(* Logix 5000 project; controller cal1632 1756-L62 rev 16.20; software revision 16.05; part 4 of 57 *)
(* tags used below, declared in another part *)
   FAULT : BOOL;
   HMI : BOOL;
   p01_ai_prs : REAL;
   p01_ai_tc : REAL;
   p01_di_edge_ctrl_estop_active : BOOL;
   p01_di_estop_1_tripped : BOOL;
   p01_di_estop_2_tripped : BOOL;
   p01_di_estop_reset : BOOL;
   p01_di_impreg_estop_active : BOOL;
   p01_di_letoff_estop_active : BOOL;
   p01_di_lof_acc_estop_active : BOOL;
   p01_di_main_hmi_estop : BOOL;
   p01_di_rope_sw_1_active : BOOL;
   p01_di_rope_sw_2_active : BOOL;
   p01_di_rope_sw_3_active : BOOL;
   p01_di_rope_sw_4_active : BOOL;
   p01_di_rope_sw_5_active : BOOL;
   p01_di_rope_sw_6_active : BOOL;
   p01_di_rope_sw_7_active : BOOL;
   p01_di_rope_sw_8_active : BOOL;
   p01_di_splice_estop_active : BOOL;
   p01_di_ts2_estop_active : BOOL;
   p01_di_winder_estop_active : BOOL;
   p01_dint_to_hmi : DINT[16];
   p01_int_from_oxidizer : INT[10];
   p01_param_master_jog_speed : REAL;
   p01_real_to_hmi : REAL[112];
   p01r02 : routine;
   p01r02_all_fans_stopped : BOOL;
   p01r02_batch_run_time_hrs : DINT;
   p01r02_do_horn : BOOL;
   p01r02_horn : BOOL;
   p01r02_timer_half_second_on : TIMER;
   p01r02_timer_second : TIMER[2];
   p01r03 : routine;
   p01r03_oxidizer_prs : SYS_SCP;
   p01r03_prs_input_max : REAL;
   p01r03_prs_input_min : REAL;
   p01r03_prs_output_max : REAL;
   p01r03_prs_output_min : REAL;
   p01r03_timer_fault : TIMER[4];
   p01r03_timer_warning : TIMER[4];
   p01r04 : routine;
   p01r04_LFL_warning : BOOL;
   p01r04_Temp_deviation_warning : BOOL;
   p01r04_timer_fault : TIMER[4];
   p01r04_timer_warning : TIMER[4];
   p01r05 : routine;
   p01r05_enc : SYS_ENC;
   p01r05_timer_fault : TIMER[4];
   p01r05_timer_warning : TIMER[4];
   p01r06 : routine;
   p01r06_timer_fault : TIMER[4];
   p01r06_timer_warning : TIMER[4];
   p01r07 : routine;
   p01r07_timer_fault : TIMER[4];
   p01r07_timer_warning : TIMER[4];
   p01r09 : routine;
   p01r09_mode_jog : BOOL;
   p01r09_mode_run : BOOL;
   p01r09_mode_thread : BOOL;
   p01r09_open_oven : BOOL;
   p01r09_pb_global_reset : BOOL;
   p01r10_fault_exists : BOOL;
   p01r10_unack_fault_ex : BOOL;
   p01r10_unack_warn_ex : BOOL;
   p01r10_warning_exists : BOOL;
   p01r12_master_ramped_speed : REAL;
   p01r13_line_running : BOOL;
   p01r13_status : DINT;
   p01r14 : routine;
   p01r14_oxidizer_heart_beat_ok : BOOL;
   p01r14_oxidizer_mass_flow : REAL;
   p11r12_Oven_auto_run_on : BOOL;
(* P01_System, continued *)

ROUTINE R03_Inputs   (* ladder *)
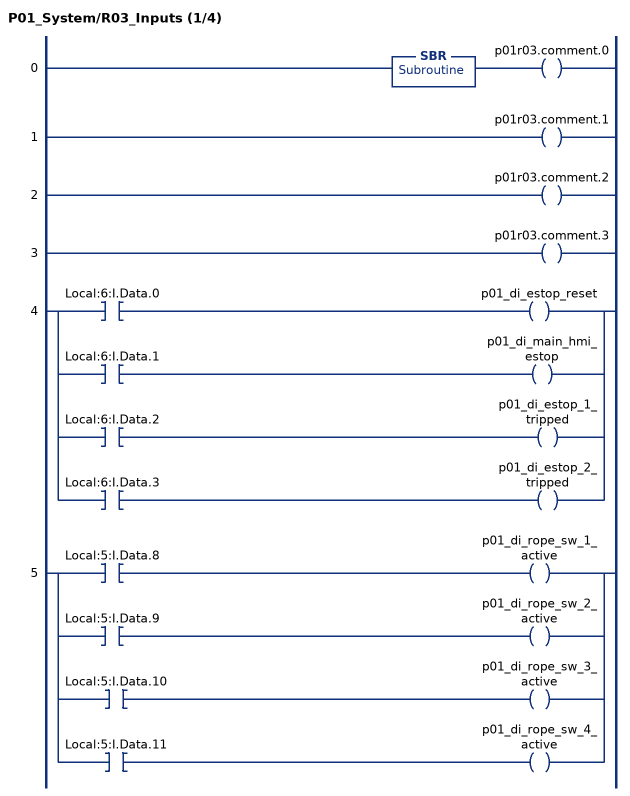
   0: SBR()OTE(p01r03.comment.0);
   1: OTE(p01r03.comment.1);
   2: OTE(p01r03.comment.2);
   3: OTE(p01r03.comment.3);
   4: [XIC(Local:6:I.Data.0) OTE(p01_di_estop_reset) ,XIC(Local:6:I.Data.1) OTE(p01_di_main_hmi_estop) ,XIC(Local:6:I.Data.2) OTE(p01_di_estop_1_tripped) ,XIC(Local:6:I.Data.3) OTE(p01_di_estop_2_tripped) ];
   5: [XIC(Local:5:I.Data.8) OTE(p01_di_rope_sw_1_active) ,XIC(Local:5:I.Data.9) OTE(p01_di_rope_sw_2_active) ,XIC(Local:5:I.Data.10) OTE(p01_di_rope_sw_3_active) ,XIC(Local:5:I.Data.11) OTE(p01_di_rope_sw_4_active) ];
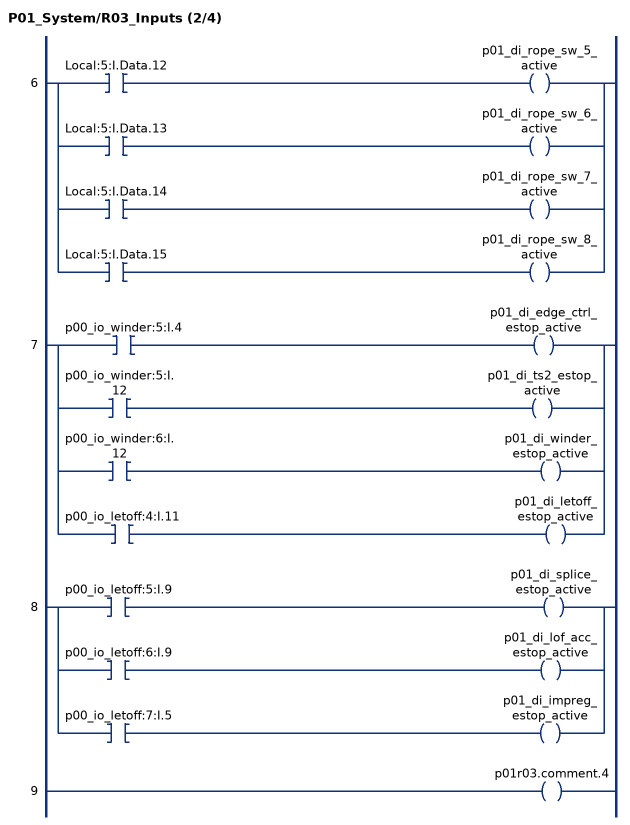
   6: [XIC(Local:5:I.Data.12) OTE(p01_di_rope_sw_5_active) ,XIC(Local:5:I.Data.13) OTE(p01_di_rope_sw_6_active) ,XIC(Local:5:I.Data.14) OTE(p01_di_rope_sw_7_active) ,XIC(Local:5:I.Data.15) OTE(p01_di_rope_sw_8_active) ];
   7: [XIC(p00_io_winder:5:I.4) OTE(p01_di_edge_ctrl_estop_active) ,XIC(p00_io_winder:5:I.12) OTE(p01_di_ts2_estop_active) ,XIC(p00_io_winder:6:I.12) OTE(p01_di_winder_estop_active) ,XIC(p00_io_letoff:4:I.11) OTE(p01_di_letoff_estop_active) ];
   8: [XIC(p00_io_letoff:5:I.9) OTE(p01_di_splice_estop_active) ,XIC(p00_io_letoff:6:I.9) OTE(p01_di_lof_acc_estop_active) ,XIC(p00_io_letoff:7:I.5) OTE(p01_di_impreg_estop_active) ];
   9: OTE(p01r03.comment.4);
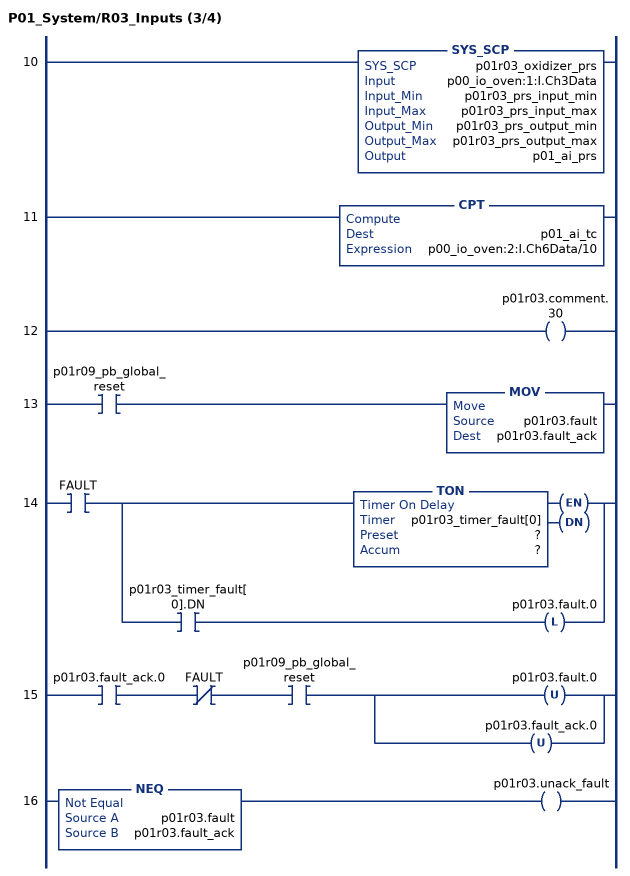
   10: SYS_SCP(p01r03_oxidizer_prs,p00_io_oven:1:I.Ch3Data,p01r03_prs_input_min,p01r03_prs_input_max,p01r03_prs_output_min,p01r03_prs_output_max,p01_ai_prs);
   11: CPT(p01_ai_tc,p00_io_oven:2:I.Ch6Data/10);
   12: OTE(p01r03.comment.30);
   13: XIC(p01r09_pb_global_reset)MOV(p01r03.fault,p01r03.fault_ack);
   14: XIC(FAULT)[TON(p01r03_timer_fault[0],?,?) ,XIC(p01r03_timer_fault[0].DN) OTL(p01r03.fault.0) ];
   15: XIC(p01r03.fault_ack.0)XIO(FAULT)XIC(p01r09_pb_global_reset)[OTU(p01r03.fault.0) ,OTU(p01r03.fault_ack.0) ];
   16: NEQ(p01r03.fault,p01r03.fault_ack)OTE(p01r03.unack_fault);
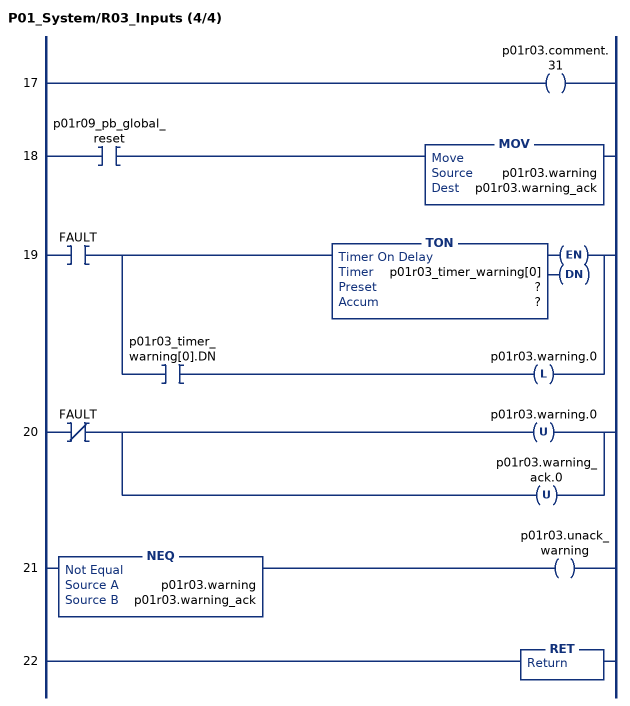
   17: OTE(p01r03.comment.31);
   18: XIC(p01r09_pb_global_reset)MOV(p01r03.warning,p01r03.warning_ack);
   19: XIC(FAULT)[TON(p01r03_timer_warning[0],?,?) ,XIC(p01r03_timer_warning[0].DN) OTL(p01r03.warning.0) ];
   20: XIO(FAULT)[OTU(p01r03.warning.0) ,OTU(p01r03.warning_ack.0) ];
   21: NEQ(p01r03.warning,p01r03.warning_ack)OTE(p01r03.unack_warning);
   22: RET();
END_ROUTINE

ROUTINE R04_Outputs   (* ladder *)
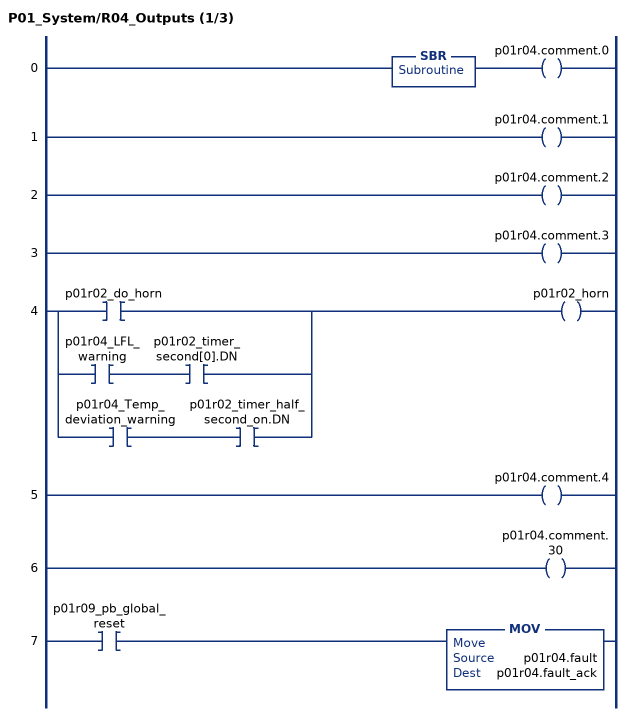
   0: SBR()OTE(p01r04.comment.0);
   1: OTE(p01r04.comment.1);
   2: OTE(p01r04.comment.2);
   3: OTE(p01r04.comment.3);
   4: [XIC(p01r02_do_horn) ,XIC(p01r04_LFL_warning) XIC(p01r02_timer_second[0].DN) ,XIC(p01r04_Temp_deviation_warning) XIC(p01r02_timer_half_second_on.DN) ]OTE(p01r02_horn);
   5: OTE(p01r04.comment.4);
   6: OTE(p01r04.comment.30);
   7: XIC(p01r09_pb_global_reset)MOV(p01r04.fault,p01r04.fault_ack);
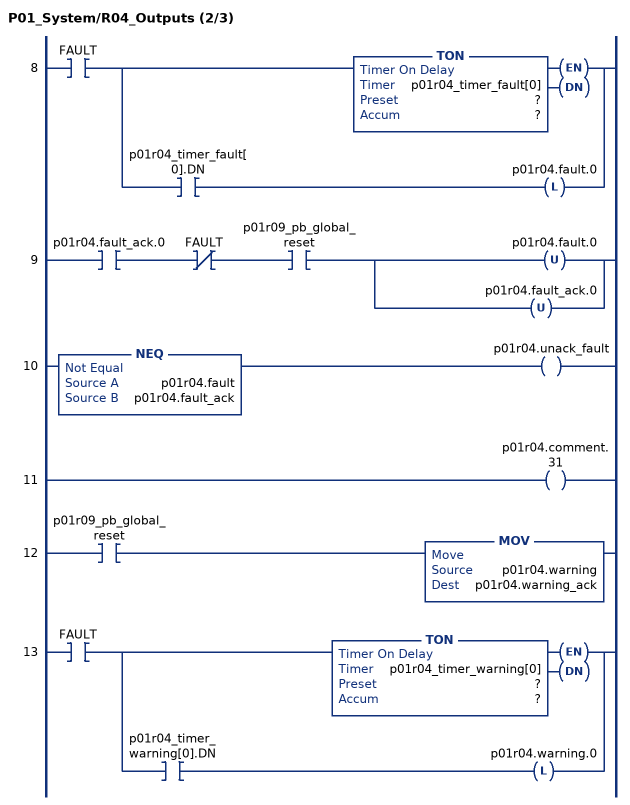
   8: XIC(FAULT)[TON(p01r04_timer_fault[0],?,?) ,XIC(p01r04_timer_fault[0].DN) OTL(p01r04.fault.0) ];
   9: XIC(p01r04.fault_ack.0)XIO(FAULT)XIC(p01r09_pb_global_reset)[OTU(p01r04.fault.0) ,OTU(p01r04.fault_ack.0) ];
   10: NEQ(p01r04.fault,p01r04.fault_ack)OTE(p01r04.unack_fault);
   11: OTE(p01r04.comment.31);
   12: XIC(p01r09_pb_global_reset)MOV(p01r04.warning,p01r04.warning_ack);
   13: XIC(FAULT)[TON(p01r04_timer_warning[0],?,?) ,XIC(p01r04_timer_warning[0].DN) OTL(p01r04.warning.0) ];
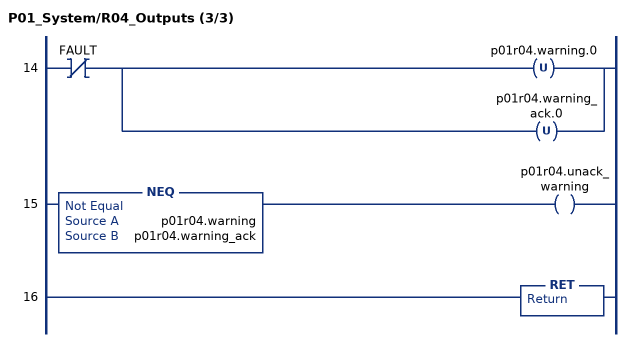
   14: XIO(FAULT)[OTU(p01r04.warning.0) ,OTU(p01r04.warning_ack.0) ];
   15: NEQ(p01r04.warning,p01r04.warning_ack)OTE(p01r04.unack_warning);
   16: RET();
END_ROUTINE

ROUTINE R05_Dint_to_HMI   (* ladder *)
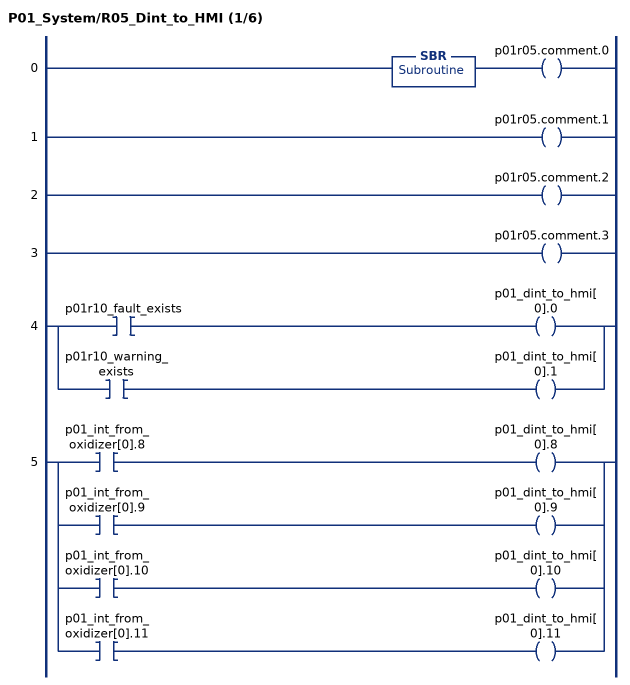
   0: SBR()OTE(p01r05.comment.0);
   1: OTE(p01r05.comment.1);
   2: OTE(p01r05.comment.2);
   3: OTE(p01r05.comment.3);
   4: [XIC(p01r10_fault_exists) OTE(p01_dint_to_hmi[0].0) ,XIC(p01r10_warning_exists) OTE(p01_dint_to_hmi[0].1) ];
   5: [XIC(p01_int_from_oxidizer[0].8) OTE(p01_dint_to_hmi[0].8) ,XIC(p01_int_from_oxidizer[0].9) OTE(p01_dint_to_hmi[0].9) ,XIC(p01_int_from_oxidizer[0].10) OTE(p01_dint_to_hmi[0].10) ,XIC(p01_int_from_oxidizer[0].11) OTE(p01_dint_to_hmi[0].11) ];
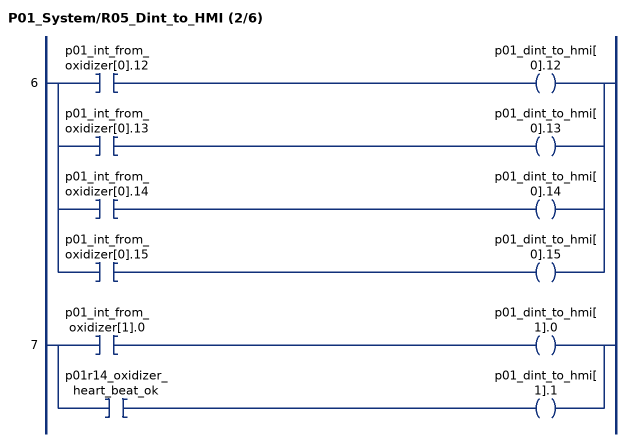
   6: [XIC(p01_int_from_oxidizer[0].12) OTE(p01_dint_to_hmi[0].12) ,XIC(p01_int_from_oxidizer[0].13) OTE(p01_dint_to_hmi[0].13) ,XIC(p01_int_from_oxidizer[0].14) OTE(p01_dint_to_hmi[0].14) ,XIC(p01_int_from_oxidizer[0].15) OTE(p01_dint_to_hmi[0].15) ];
   7: [XIC(p01_int_from_oxidizer[1].0) OTE(p01_dint_to_hmi[1].0) ,XIC(p01r14_oxidizer_heart_beat_ok) OTE(p01_dint_to_hmi[1].1) ];
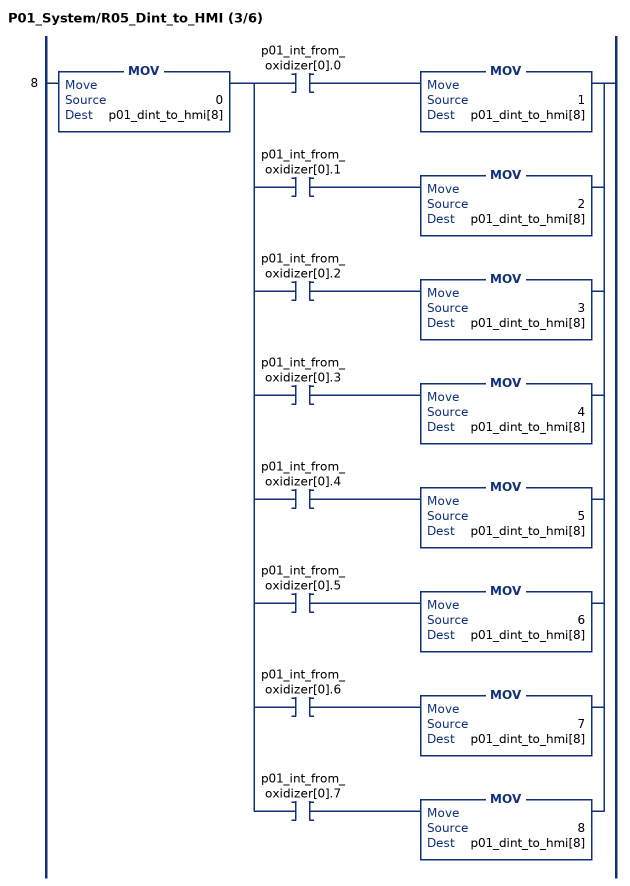
   8: MOV(0,p01_dint_to_hmi[8])[XIC(p01_int_from_oxidizer[0].0) MOV(1,p01_dint_to_hmi[8]) ,XIC(p01_int_from_oxidizer[0].1) MOV(2,p01_dint_to_hmi[8]) ,XIC(p01_int_from_oxidizer[0].2) MOV(3,p01_dint_to_hmi[8]) ,XIC(p01_int_from_oxidizer[0].3) MOV(4,p01_dint_to_hmi[8]) ,XIC(p01_int_from_oxidizer[0].4) MOV(5,p01_dint_to_hmi[8]) ,XIC(p01_int_from_oxidizer[0].5) MOV(6,p01_dint_to_hmi[8]) ,XIC(p01_int_from_oxidizer[0].6) MOV(7,p01_dint_to_hmi[8]) ,XIC(p01_int_from_oxidizer[0].7) MOV(8,p01_dint_to_hmi[8]) ];
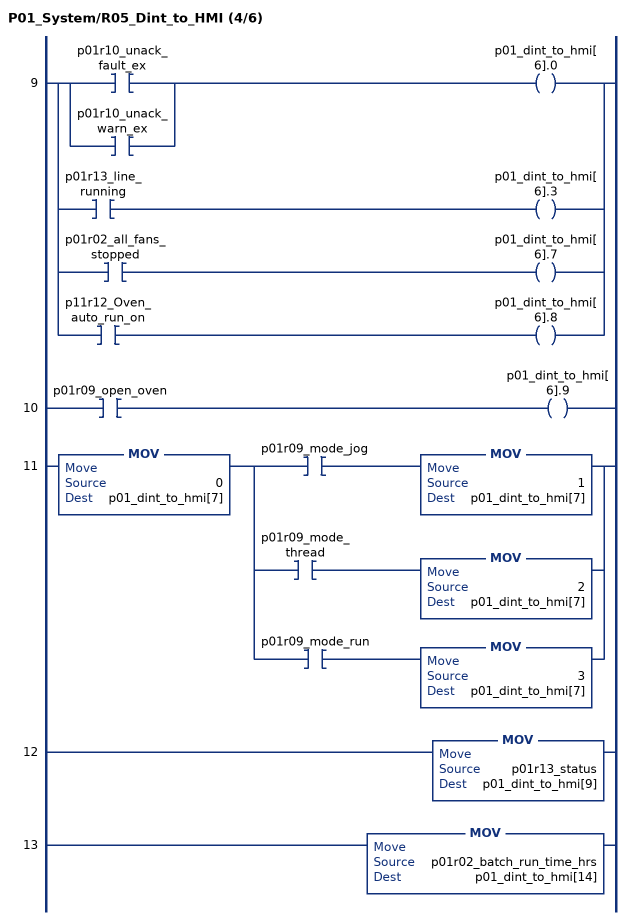
   9: [[XIC(p01r10_unack_fault_ex) ,XIC(p01r10_unack_warn_ex) ] OTE(p01_dint_to_hmi[6].0) ,XIC(p01r13_line_running) OTE(p01_dint_to_hmi[6].3) ,XIC(p01r02_all_fans_stopped) OTE(p01_dint_to_hmi[6].7) ,XIC(p11r12_Oven_auto_run_on) OTE(p01_dint_to_hmi[6].8) ];
   10: XIC(p01r09_open_oven)OTE(p01_dint_to_hmi[6].9);
   11: MOV(0,p01_dint_to_hmi[7])[XIC(p01r09_mode_jog) MOV(1,p01_dint_to_hmi[7]) ,XIC(p01r09_mode_thread) MOV(2,p01_dint_to_hmi[7]) ,XIC(p01r09_mode_run) MOV(3,p01_dint_to_hmi[7]) ];
   12: MOV(p01r13_status,p01_dint_to_hmi[9]);
   13: MOV(p01r02_batch_run_time_hrs,p01_dint_to_hmi[14]);
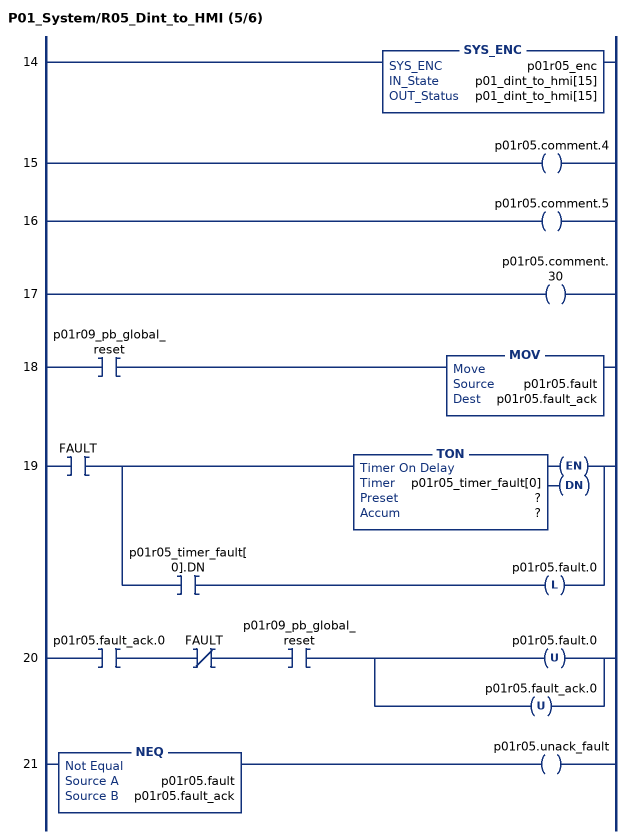
   14: SYS_ENC(p01r05_enc,p01_dint_to_hmi[15],p01_dint_to_hmi[15]);
   15: OTE(p01r05.comment.4);
   16: OTE(p01r05.comment.5);
   17: OTE(p01r05.comment.30);
   18: XIC(p01r09_pb_global_reset)MOV(p01r05.fault,p01r05.fault_ack);
   19: XIC(FAULT)[TON(p01r05_timer_fault[0],?,?) ,XIC(p01r05_timer_fault[0].DN) OTL(p01r05.fault.0) ];
   20: XIC(p01r05.fault_ack.0)XIO(FAULT)XIC(p01r09_pb_global_reset)[OTU(p01r05.fault.0) ,OTU(p01r05.fault_ack.0) ];
   21: NEQ(p01r05.fault,p01r05.fault_ack)OTE(p01r05.unack_fault);
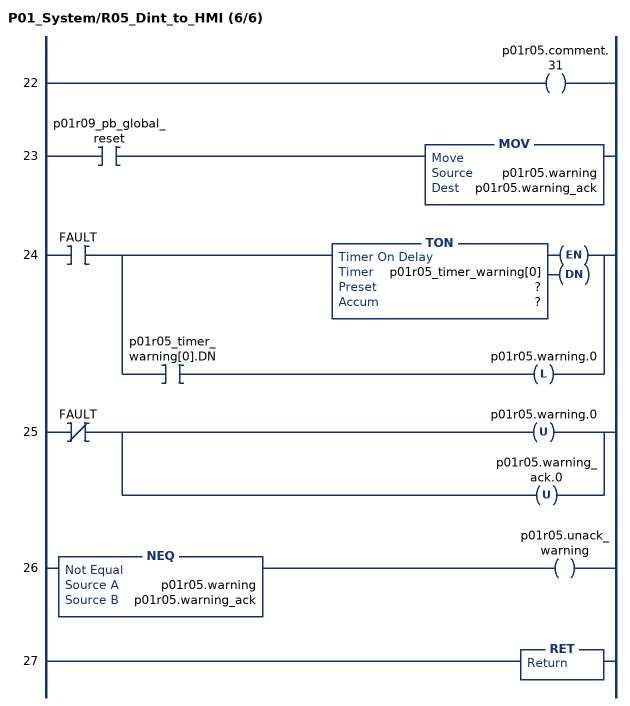
   22: OTE(p01r05.comment.31);
   23: XIC(p01r09_pb_global_reset)MOV(p01r05.warning,p01r05.warning_ack);
   24: XIC(FAULT)[TON(p01r05_timer_warning[0],?,?) ,XIC(p01r05_timer_warning[0].DN) OTL(p01r05.warning.0) ];
   25: XIO(FAULT)[OTU(p01r05.warning.0) ,OTU(p01r05.warning_ack.0) ];
   26: NEQ(p01r05.warning,p01r05.warning_ack)OTE(p01r05.unack_warning);
   27: RET();
END_ROUTINE

ROUTINE R06_Real_to_HMI   (* ladder *)
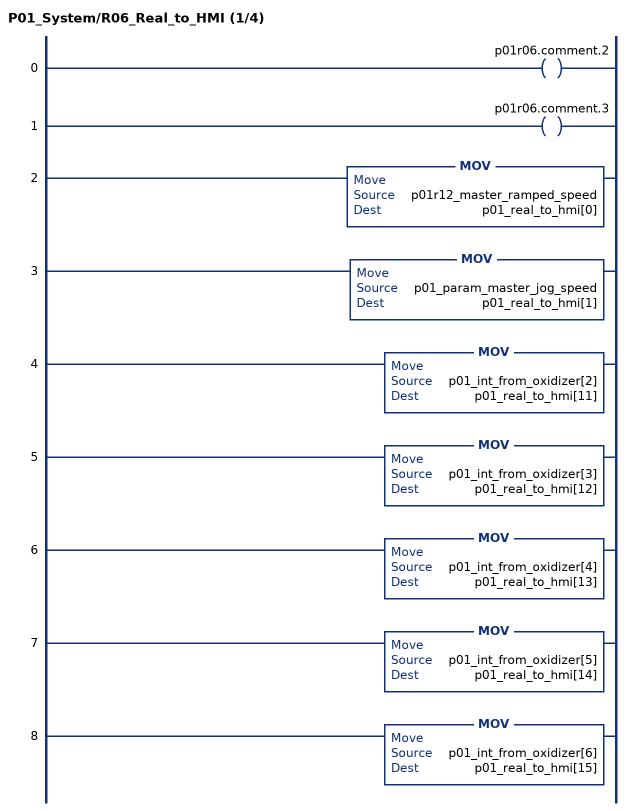
   0: OTE(p01r06.comment.2);
   1: OTE(p01r06.comment.3);
   2: MOV(p01r12_master_ramped_speed,p01_real_to_hmi[0]);
   3: MOV(p01_param_master_jog_speed,p01_real_to_hmi[1]);
   4: MOV(p01_int_from_oxidizer[2],p01_real_to_hmi[11]);
   5: MOV(p01_int_from_oxidizer[3],p01_real_to_hmi[12]);
   6: MOV(p01_int_from_oxidizer[4],p01_real_to_hmi[13]);
   7: MOV(p01_int_from_oxidizer[5],p01_real_to_hmi[14]);
   8: MOV(p01_int_from_oxidizer[6],p01_real_to_hmi[15]);
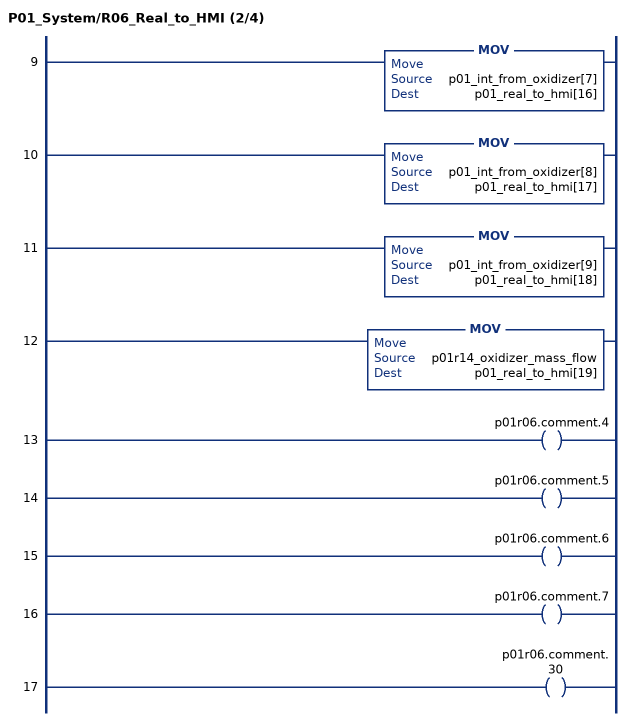
   9: MOV(p01_int_from_oxidizer[7],p01_real_to_hmi[16]);
   10: MOV(p01_int_from_oxidizer[8],p01_real_to_hmi[17]);
   11: MOV(p01_int_from_oxidizer[9],p01_real_to_hmi[18]);
   12: MOV(p01r14_oxidizer_mass_flow,p01_real_to_hmi[19]);
   13: OTE(p01r06.comment.4);
   14: OTE(p01r06.comment.5);
   15: OTE(p01r06.comment.6);
   16: OTE(p01r06.comment.7);
   17: OTE(p01r06.comment.30);
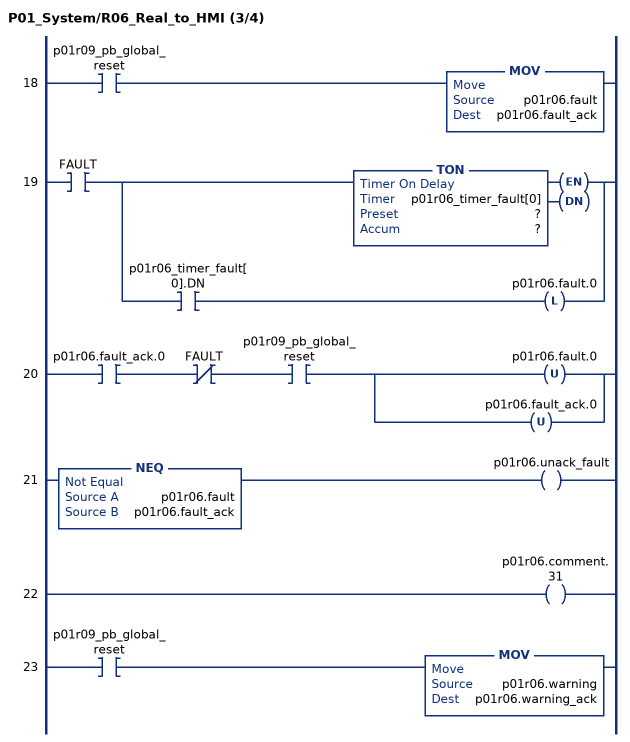
   18: XIC(p01r09_pb_global_reset)MOV(p01r06.fault,p01r06.fault_ack);
   19: XIC(FAULT)[TON(p01r06_timer_fault[0],?,?) ,XIC(p01r06_timer_fault[0].DN) OTL(p01r06.fault.0) ];
   20: XIC(p01r06.fault_ack.0)XIO(FAULT)XIC(p01r09_pb_global_reset)[OTU(p01r06.fault.0) ,OTU(p01r06.fault_ack.0) ];
   21: NEQ(p01r06.fault,p01r06.fault_ack)OTE(p01r06.unack_fault);
   22: OTE(p01r06.comment.31);
   23: XIC(p01r09_pb_global_reset)MOV(p01r06.warning,p01r06.warning_ack);
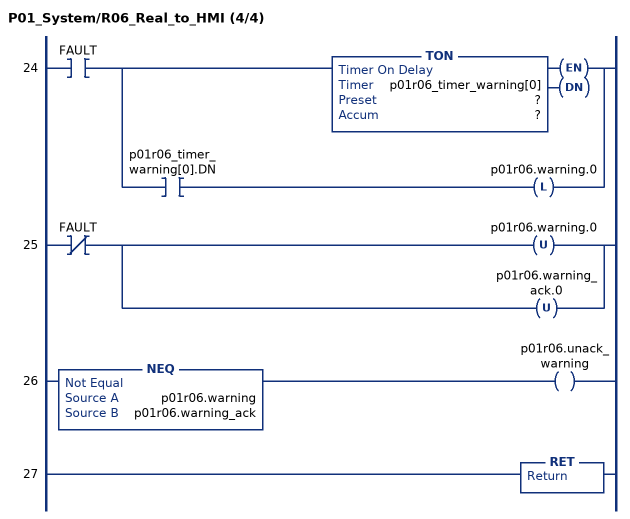
   24: XIC(FAULT)[TON(p01r06_timer_warning[0],?,?) ,XIC(p01r06_timer_warning[0].DN) OTL(p01r06.warning.0) ];
   25: XIO(FAULT)[OTU(p01r06.warning.0) ,OTU(p01r06.warning_ack.0) ];
   26: NEQ(p01r06.warning,p01r06.warning_ack)OTE(p01r06.unack_warning);
   27: RET();
END_ROUTINE

ROUTINE R07_Alarms   (* ladder *)
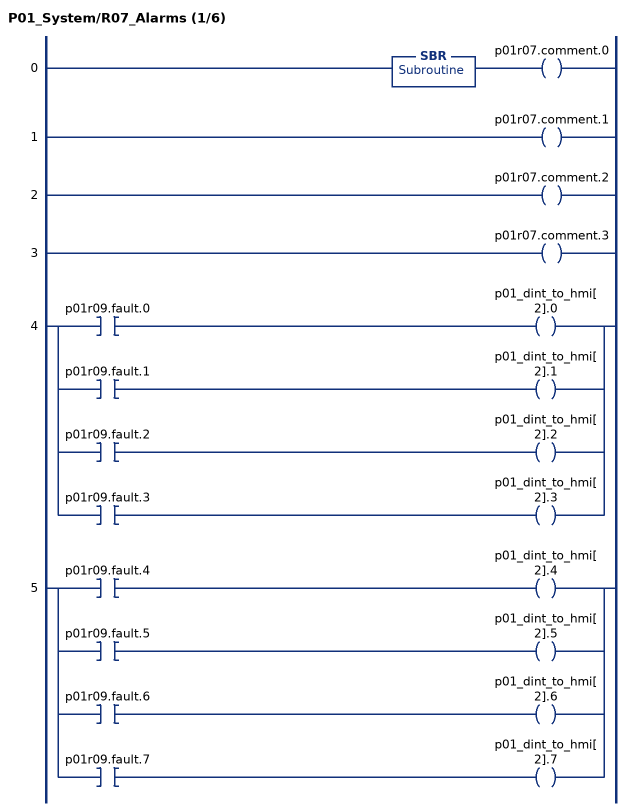
   0: SBR()OTE(p01r07.comment.0);
   1: OTE(p01r07.comment.1);
   2: OTE(p01r07.comment.2);
   3: OTE(p01r07.comment.3);
   4: [XIC(p01r09.fault.0) OTE(p01_dint_to_hmi[2].0) ,XIC(p01r09.fault.1) OTE(p01_dint_to_hmi[2].1) ,XIC(p01r09.fault.2) OTE(p01_dint_to_hmi[2].2) ,XIC(p01r09.fault.3) OTE(p01_dint_to_hmi[2].3) ];
   5: [XIC(p01r09.fault.4) OTE(p01_dint_to_hmi[2].4) ,XIC(p01r09.fault.5) OTE(p01_dint_to_hmi[2].5) ,XIC(p01r09.fault.6) OTE(p01_dint_to_hmi[2].6) ,XIC(p01r09.fault.7) OTE(p01_dint_to_hmi[2].7) ];
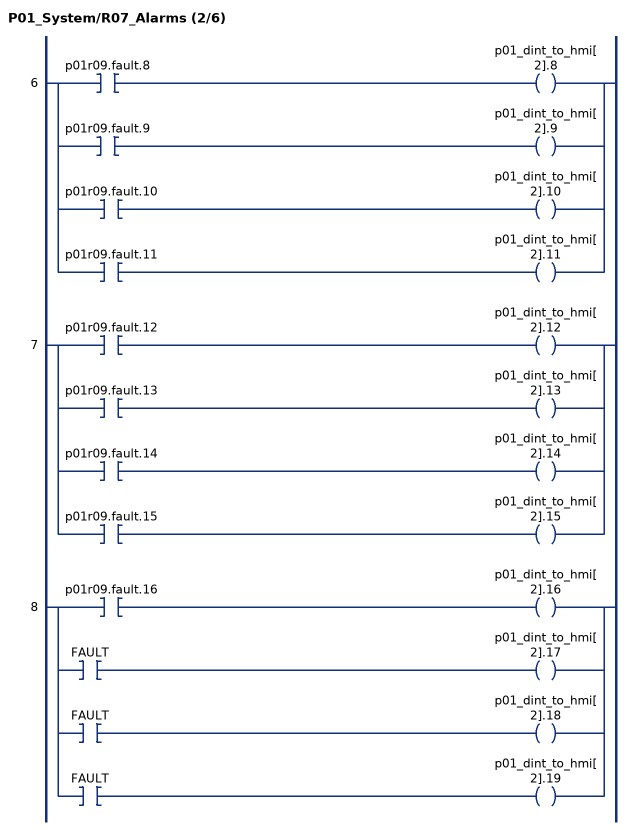
   6: [XIC(p01r09.fault.8) OTE(p01_dint_to_hmi[2].8) ,XIC(p01r09.fault.9) OTE(p01_dint_to_hmi[2].9) ,XIC(p01r09.fault.10) OTE(p01_dint_to_hmi[2].10) ,XIC(p01r09.fault.11) OTE(p01_dint_to_hmi[2].11) ];
   7: [XIC(p01r09.fault.12) OTE(p01_dint_to_hmi[2].12) ,XIC(p01r09.fault.13) OTE(p01_dint_to_hmi[2].13) ,XIC(p01r09.fault.14) OTE(p01_dint_to_hmi[2].14) ,XIC(p01r09.fault.15) OTE(p01_dint_to_hmi[2].15) ];
   8: [XIC(p01r09.fault.16) OTE(p01_dint_to_hmi[2].16) ,XIC(FAULT) OTE(p01_dint_to_hmi[2].17) ,XIC(FAULT) OTE(p01_dint_to_hmi[2].18) ,XIC(FAULT) OTE(p01_dint_to_hmi[2].19) ];
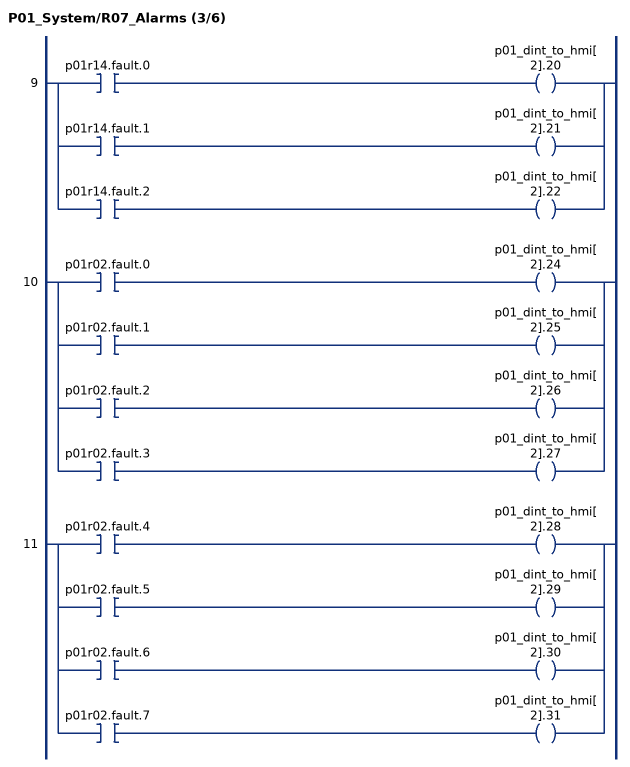
   9: [XIC(p01r14.fault.0) OTE(p01_dint_to_hmi[2].20) ,XIC(p01r14.fault.1) OTE(p01_dint_to_hmi[2].21) ,XIC(p01r14.fault.2) OTE(p01_dint_to_hmi[2].22) ];
   10: [XIC(p01r02.fault.0) OTE(p01_dint_to_hmi[2].24) ,XIC(p01r02.fault.1) OTE(p01_dint_to_hmi[2].25) ,XIC(p01r02.fault.2) OTE(p01_dint_to_hmi[2].26) ,XIC(p01r02.fault.3) OTE(p01_dint_to_hmi[2].27) ];
   11: [XIC(p01r02.fault.4) OTE(p01_dint_to_hmi[2].28) ,XIC(p01r02.fault.5) OTE(p01_dint_to_hmi[2].29) ,XIC(p01r02.fault.6) OTE(p01_dint_to_hmi[2].30) ,XIC(p01r02.fault.7) OTE(p01_dint_to_hmi[2].31) ];
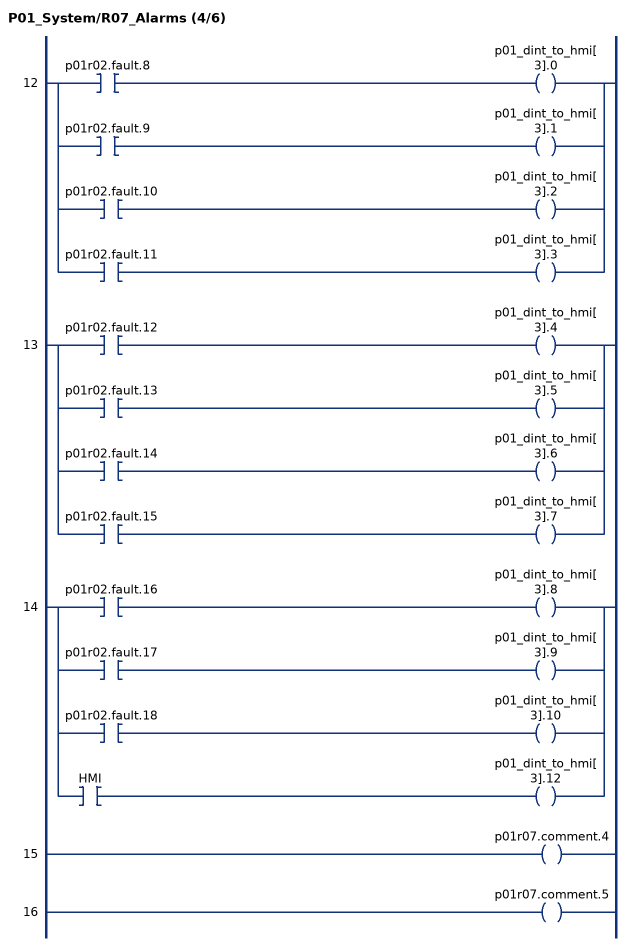
   12: [XIC(p01r02.fault.8) OTE(p01_dint_to_hmi[3].0) ,XIC(p01r02.fault.9) OTE(p01_dint_to_hmi[3].1) ,XIC(p01r02.fault.10) OTE(p01_dint_to_hmi[3].2) ,XIC(p01r02.fault.11) OTE(p01_dint_to_hmi[3].3) ];
   13: [XIC(p01r02.fault.12) OTE(p01_dint_to_hmi[3].4) ,XIC(p01r02.fault.13) OTE(p01_dint_to_hmi[3].5) ,XIC(p01r02.fault.14) OTE(p01_dint_to_hmi[3].6) ,XIC(p01r02.fault.15) OTE(p01_dint_to_hmi[3].7) ];
   14: [XIC(p01r02.fault.16) OTE(p01_dint_to_hmi[3].8) ,XIC(p01r02.fault.17) OTE(p01_dint_to_hmi[3].9) ,XIC(p01r02.fault.18) OTE(p01_dint_to_hmi[3].10) ,XIC(HMI) OTE(p01_dint_to_hmi[3].12) ];
   15: OTE(p01r07.comment.4);
   16: OTE(p01r07.comment.5);
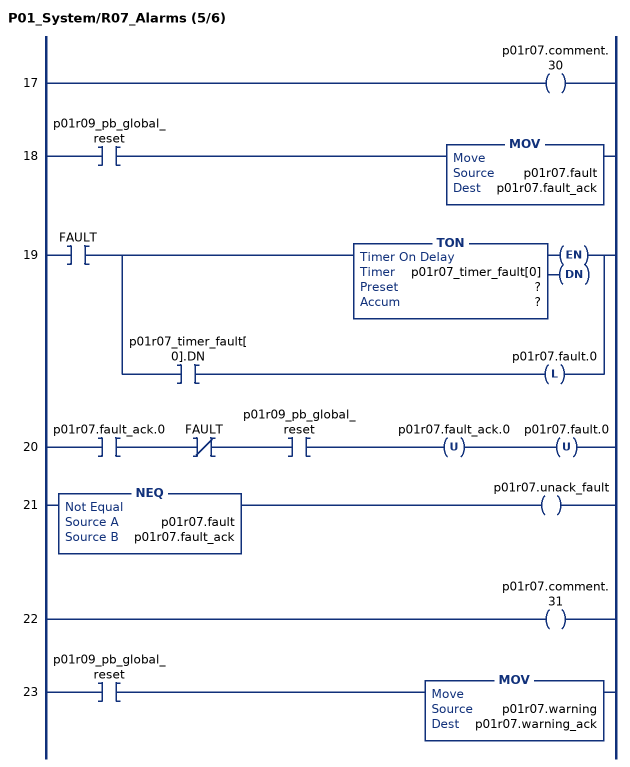
   17: OTE(p01r07.comment.30);
   18: XIC(p01r09_pb_global_reset)MOV(p01r07.fault,p01r07.fault_ack);
   19: XIC(FAULT)[TON(p01r07_timer_fault[0],?,?) ,XIC(p01r07_timer_fault[0].DN) OTL(p01r07.fault.0) ];
   20: XIC(p01r07.fault_ack.0)XIO(FAULT)XIC(p01r09_pb_global_reset)OTU(p01r07.fault_ack.0)OTU(p01r07.fault.0);
   21: NEQ(p01r07.fault,p01r07.fault_ack)OTE(p01r07.unack_fault);
   22: OTE(p01r07.comment.31);
   23: XIC(p01r09_pb_global_reset)MOV(p01r07.warning,p01r07.warning_ack);
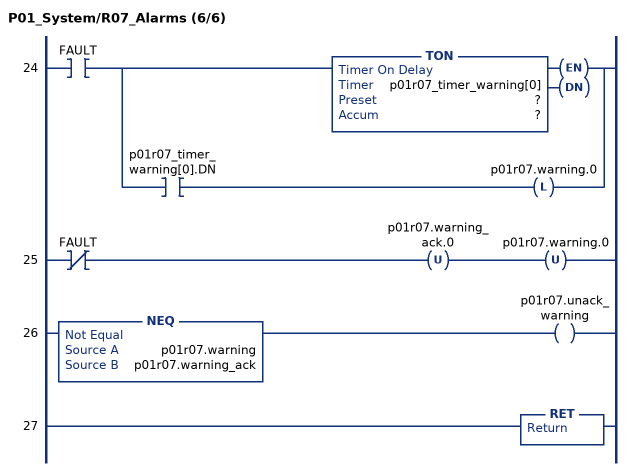
   24: XIC(FAULT)[TON(p01r07_timer_warning[0],?,?) ,XIC(p01r07_timer_warning[0].DN) OTL(p01r07.warning.0) ];
   25: XIO(FAULT)OTU(p01r07.warning_ack.0)OTU(p01r07.warning.0);
   26: NEQ(p01r07.warning,p01r07.warning_ack)OTE(p01r07.unack_warning);
   27: RET();
END_ROUTINE
